(* IEC 61131-3 sources: plc_generation_empirical_study/datasets/task_bank_c06_bounded_runtime_v0_3/tasks/C06_U14_lean_composite/negative_control, 1 file *)

(* ---- NC1.st ---- *)
FUNCTION_BLOCK C06_U14_lean_composite
VAR_INPUT
    A_Item : BOOL;
    A_Reset : BOOL;
    A_Target : INT;
    A_Enable : BOOL;
    B_AutoMode : BOOL;
    B_AutoDemand : BOOL;
    B_ManualDemand : BOOL;
    B_SafetyOK : BOOL;
    B_Inhibit : BOOL;
    SubsystemBEnable : BOOL;
    CrossReset : BOOL;
END_VAR
VAR_OUTPUT
    A_Count : INT;
    A_BatchDone : BOOL;
    A_Accepted : BOOL;
    B_Command : BOOL;
    B_Blocked : BOOL;
    CrossReady : BOOL;
    CrossBlocked : BOOL;
END_VAR
VAR
    A_PrevItem : BOOL := FALSE;
END_VAR

A_Accepted := FALSE;
IF A_Reset THEN
    A_Count := 0;
ELSIF A_Enable AND A_Item AND (NOT A_PrevItem) AND (A_Count < A_Target) THEN
    A_Count := A_Count + 1;
    A_Accepted := TRUE;
END_IF;
A_BatchDone := A_Count >= A_Target;
A_PrevItem := A_Item;

IF CrossReset THEN
    CrossReady := FALSE;
ELSIF A_BatchDone THEN
    CrossReady := TRUE;
END_IF;
CrossBlocked := FALSE;

IF SubsystemBEnable AND CrossReady THEN
    B_Command := ((B_AutoMode AND B_AutoDemand) OR ((NOT B_AutoMode) AND B_ManualDemand))
               AND B_SafetyOK AND (NOT B_Inhibit);
    B_Blocked := ((B_AutoMode AND B_AutoDemand) OR ((NOT B_AutoMode) AND B_ManualDemand))
               AND ((NOT B_SafetyOK) OR B_Inhibit);
ELSE
    B_Command := FALSE;
    B_Blocked := FALSE;
END_IF;

END_FUNCTION_BLOCK
